// Mitsubishi GX Works2 project: 3개 논리회로 (XOR)   PLC: Q02/Q02H

PROGRAM MAIN
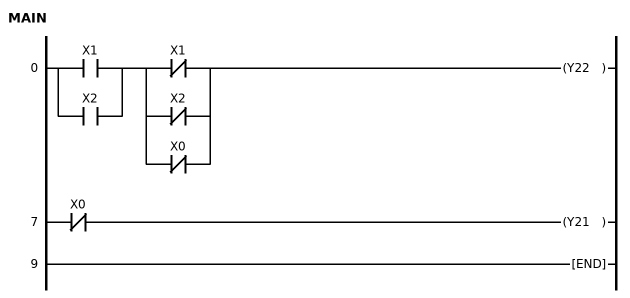
0     LD      X1
      OR      X2
      LDI     X1
      ORI     X2
      ORI     X0
      ANB
      OUT     Y22
7     LDI     X0
      OUT     Y21
9     END
END_PROGRAM
